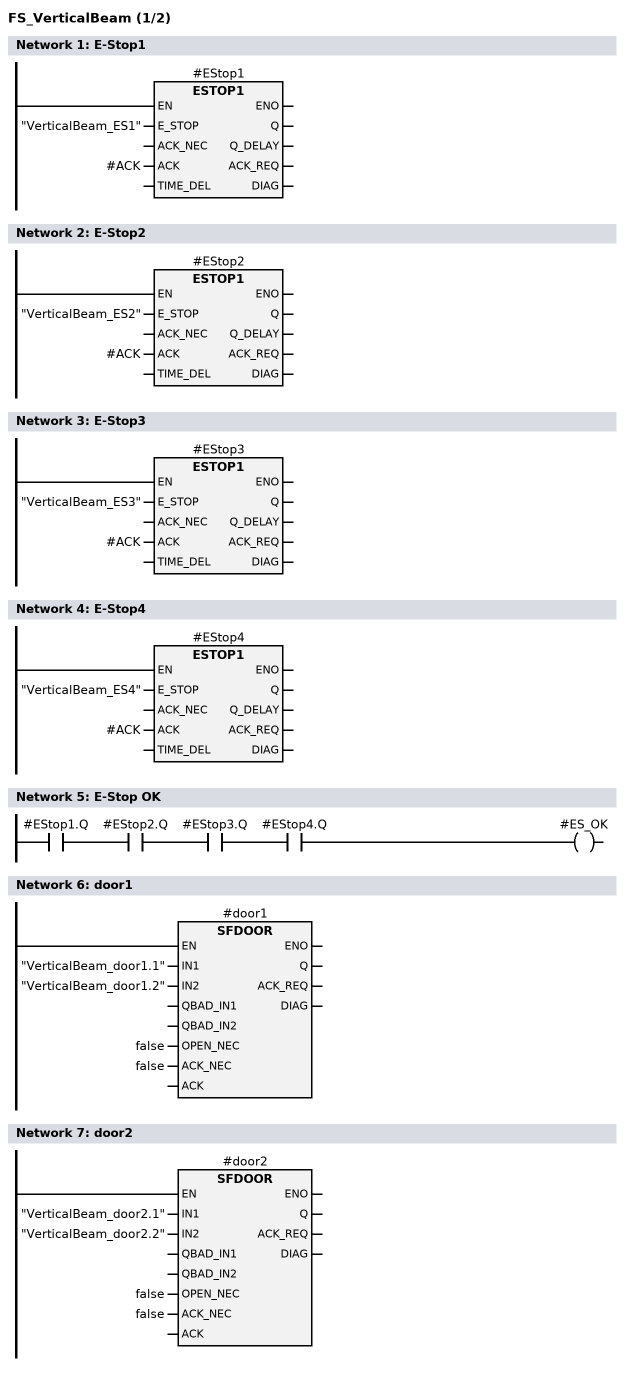
   RUNG wire#powerrail
      #EStop1.ESTOP1(E_STOP := "VerticalBeam_ES1", ACK_NEC :=, ACK := #ACK, TIME_DEL :=, Q =>, Q_DELAY =>, ACK_REQ =>, DIAG =>)
   END_RUNG
   // the same network as SCL:
   #EStop1(E_STOP := "VerticalBeam_ES1", ACK := #ACK);   // ESTOP1
END_REGION

REGION Network 2: E-Stop2
   RUNG wire#powerrail
      #EStop2.ESTOP1(E_STOP := "VerticalBeam_ES2", ACK_NEC :=, ACK := #ACK, TIME_DEL :=, Q =>, Q_DELAY =>, ACK_REQ =>, DIAG =>)
   END_RUNG
   // the same network as SCL:
   #EStop2(E_STOP := "VerticalBeam_ES2", ACK := #ACK);   // ESTOP1
END_REGION

REGION Network 3: E-Stop3
   RUNG wire#powerrail
      #EStop3.ESTOP1(E_STOP := "VerticalBeam_ES3", ACK_NEC :=, ACK := #ACK, TIME_DEL :=, Q =>, Q_DELAY =>, ACK_REQ =>, DIAG =>)
   END_RUNG
   // the same network as SCL:
   #EStop3(E_STOP := "VerticalBeam_ES3", ACK := #ACK);   // ESTOP1
END_REGION

REGION Network 4: E-Stop4
   RUNG wire#powerrail
      #EStop4.ESTOP1(E_STOP := "VerticalBeam_ES4", ACK_NEC :=, ACK := #ACK, TIME_DEL :=, Q =>, Q_DELAY =>, ACK_REQ =>, DIAG =>)
   END_RUNG
   // the same network as SCL:
   #EStop4(E_STOP := "VerticalBeam_ES4", ACK := #ACK);   // ESTOP1
END_REGION

REGION Network 5: E-Stop OK
   RUNG wire#powerrail
      Contact( #EStop1.Q )
      Contact( #EStop2.Q )
      Contact( #EStop3.Q )
      Contact( #EStop4.Q )
      Coil( #ES_OK )
   END_RUNG
   // the same network as SCL:
   #ES_OK := #EStop1.Q AND #EStop2.Q AND #EStop3.Q AND #EStop4.Q;
END_REGION

REGION Network 6: door1
   RUNG wire#powerrail
      #door1.SFDOOR(IN1 := "VerticalBeam_door1.1", IN2 := "VerticalBeam_door1.2", QBAD_IN1 :=, QBAD_IN2 :=, OPEN_NEC := false, ACK_NEC := false, ACK :=, Q =>, ACK_REQ =>, DIAG =>)
   END_RUNG
   // the same network as SCL:
   #door1(IN1 := "VerticalBeam_door1.1", IN2 := "VerticalBeam_door1.2", OPEN_NEC := false, ACK_NEC := false);   // SFDOOR
END_REGION

REGION Network 7: door2
   RUNG wire#powerrail
      #door2.SFDOOR(IN1 := "VerticalBeam_door2.1", IN2 := "VerticalBeam_door2.2", QBAD_IN1 :=, QBAD_IN2 :=, OPEN_NEC := false, ACK_NEC := false, ACK :=, Q =>, ACK_REQ =>, DIAG =>)
   END_RUNG
   // the same network as SCL:
   #door2(IN1 := "VerticalBeam_door2.1", IN2 := "VerticalBeam_door2.2", OPEN_NEC := false, ACK_NEC := false);   // SFDOOR
END_REGION

REGION Network 8: Key
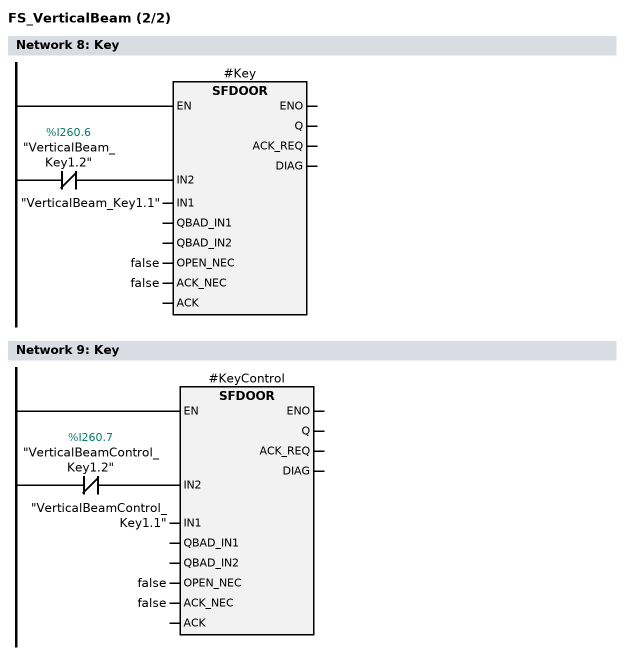
   RUNG wire#powerrail
      #Key.SFDOOR(IN2 := wire#w1, IN1 := "VerticalBeam_Key1.1", QBAD_IN1 :=, QBAD_IN2 :=, OPEN_NEC := false, ACK_NEC := false, ACK :=, Q =>, ACK_REQ =>, DIAG =>)
   END_RUNG
   RUNG wire#powerrail
      I_Contact( "VerticalBeam_Key1.2" )
   END_RUNG wire#w1
   // the same network as SCL:
   #Key(IN2 := NOT "VerticalBeam_Key1.2", IN1 := "VerticalBeam_Key1.1", OPEN_NEC := false, ACK_NEC := false);   // SFDOOR
END_REGION

REGION Network 9: Key
   RUNG wire#powerrail
      #KeyControl.SFDOOR(IN2 := wire#w1, IN1 := "VerticalBeamControl_Key1.1", QBAD_IN1 :=, QBAD_IN2 :=, OPEN_NEC := false, ACK_NEC := false, ACK :=, Q =>, ACK_REQ =>, DIAG =>)
   END_RUNG
   RUNG wire#powerrail
      I_Contact( "VerticalBeamControl_Key1.2" )
   END_RUNG wire#w1
   // the same network as SCL:
   #KeyControl(IN2 := NOT "VerticalBeamControl_Key1.2",   // SFDOOR
               IN1 := "VerticalBeamControl_Key1.1",
               OPEN_NEC := false,
               ACK_NEC := false);
END_REGION
END_FUNCTION_BLOCK

FUNCTION "F_ChannelDia" : Void   // FC2, F_LAD
{ S7_Optimized_Access := 'TRUE' }
VERSION : 0.1
// stored: AutoNumber true, IsIECCheckEnabled false, UDAEnableTagReadback false
   VAR_INPUT
      PASS_OUT : Bool;
      QBAD : Bool;
      ACK_REQ : Bool;
      Channel0_ValueStatus : Bool;
      Channel1_ValueStatus : Bool;
      Channel2_ValueStatus : Bool;
      Channel3_ValueStatus : Bool;
      Channel4_ValueStatus : Bool;
      Channel5_ValueStatus : Bool;
      Channel6_ValueStatus : Bool;
      Channel7_ValueStatus : Bool;
   END_VAR
   VAR_OUTPUT
      FIODia : "FIODia";
   END_VAR
   VAR_TEMP   // added for the SCL form of the ladder/FBD networks
      _w1 : Bool;
   END_VAR
BEGIN

REGION Network 1: 模块钝化
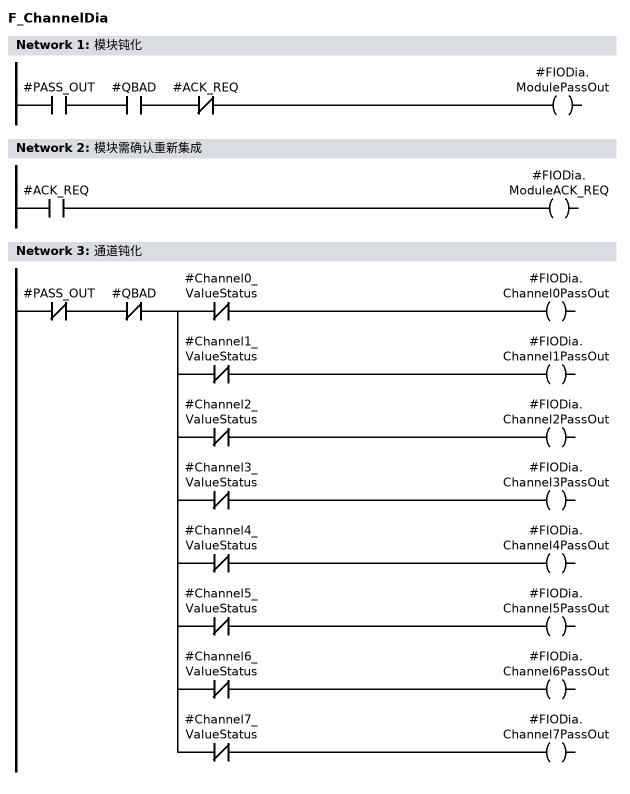
   RUNG wire#powerrail
      Contact( #PASS_OUT )
      Contact( #QBAD )
      I_Contact( #ACK_REQ )
      Coil( #FIODia.ModulePassOut )
   END_RUNG
   // the same network as SCL:
   #FIODia.ModulePassOut := #PASS_OUT AND #QBAD AND NOT #ACK_REQ;
END_REGION

REGION Network 2: 模块需确认重新集成
   RUNG wire#powerrail
      Contact( #ACK_REQ )
      Coil( #FIODia.ModuleACK_REQ )
   END_RUNG
   // the same network as SCL:
   #FIODia.ModuleACK_REQ := #ACK_REQ;
END_REGION

REGION Network 3: 通道钝化
   RUNG wire#powerrail
      I_Contact( #PASS_OUT )
      I_Contact( #QBAD )
      wire#w1
      I_Contact( #Channel0_ValueStatus )
      Coil( #FIODia.Channel0PassOut )
   END_RUNG
   RUNG wire#w1
      I_Contact( #Channel1_ValueStatus )
      Coil( #FIODia.Channel1PassOut )
   END_RUNG
   RUNG wire#w1
      I_Contact( #Channel2_ValueStatus )
      Coil( #FIODia.Channel2PassOut )
   END_RUNG
   RUNG wire#w1
      I_Contact( #Channel3_ValueStatus )
      Coil( #FIODia.Channel3PassOut )
   END_RUNG
   RUNG wire#w1
      I_Contact( #Channel4_ValueStatus )
      Coil( #FIODia.Channel4PassOut )
   END_RUNG
   RUNG wire#w1
      I_Contact( #Channel5_ValueStatus )
      Coil( #FIODia.Channel5PassOut )
   END_RUNG
   RUNG wire#w1
      I_Contact( #Channel6_ValueStatus )
      Coil( #FIODia.Channel6PassOut )
   END_RUNG
   RUNG wire#w1
      I_Contact( #Channel7_ValueStatus )
      Coil( #FIODia.Channel7PassOut )
   END_RUNG
   // the same network as SCL:
   #_w1 := NOT #PASS_OUT AND NOT #QBAD;
   #FIODia.Channel0PassOut := #_w1 AND NOT #Channel0_ValueStatus;
   #FIODia.Channel1PassOut := #_w1 AND NOT #Channel1_ValueStatus;
   #FIODia.Channel2PassOut := #_w1 AND NOT #Channel2_ValueStatus;
   #FIODia.Channel3PassOut := #_w1 AND NOT #Channel3_ValueStatus;
   #FIODia.Channel4PassOut := #_w1 AND NOT #Channel4_ValueStatus;
   #FIODia.Channel5PassOut := #_w1 AND NOT #Channel5_ValueStatus;
   #FIODia.Channel6PassOut := #_w1 AND NOT #Channel6_ValueStatus;
   #FIODia.Channel7PassOut := #_w1 AND NOT #Channel7_ValueStatus;
END_REGION
END_FUNCTION

FUNCTION "Interlock" : Void   // FC1, F_LAD
{ S7_Optimized_Access := 'TRUE' }
VERSION : 0.1
// stored: AutoNumber true, IsIECCheckEnabled false, UDAEnableTagReadback false
   VAR_INPUT
      Room1_Interlock : Bool;
      Room2_Interlock : Bool;
      ACC_Interlock : Bool;
      VerticalBeam_Interlock : Bool;
      "E-stop" : Bool;
   END_VAR
BEGIN

REGION Network 1
   // 暂未考虑模块钝化和通道钝化情况
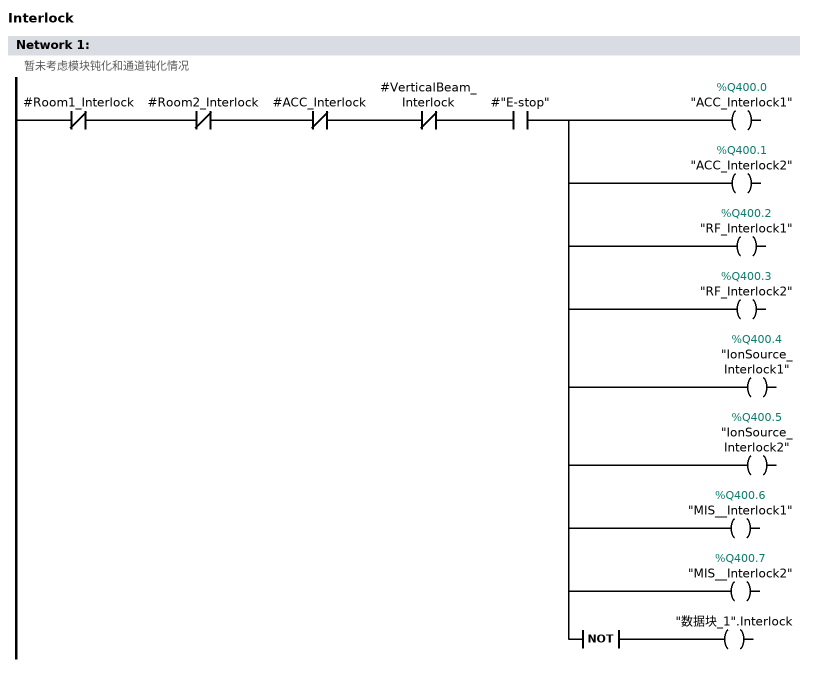
   RUNG wire#powerrail
      I_Contact( #Room1_Interlock )
      I_Contact( #Room2_Interlock )
      I_Contact( #ACC_Interlock )
      I_Contact( #VerticalBeam_Interlock )
      Contact( #"E-stop" )
      wire#w1
      Coil( "ACC_Interlock1" )
   END_RUNG
   RUNG wire#w1
      Coil( "ACC_Interlock2" )
   END_RUNG
   RUNG wire#w1
      Coil( "RF_Interlock1" )
   END_RUNG
   RUNG wire#w1
      Coil( "RF_Interlock2" )
   END_RUNG
   RUNG wire#w1
      Coil( "IonSource_Interlock1" )
   END_RUNG
   RUNG wire#w1
      Coil( "IonSource_Interlock2" )
   END_RUNG
   RUNG wire#w1
      Coil( "MIS__Interlock1" )
   END_RUNG
   RUNG wire#w1
      Coil( "MIS__Interlock2" )
   END_RUNG
   RUNG wire#w1
      Not()
      Coil( "数据块_1".Interlock )
   END_RUNG
   // the same network as SCL:
   "ACC_Interlock1" := NOT #Room1_Interlock AND NOT #Room2_Interlock AND NOT #ACC_Interlock AND NOT #VerticalBeam_Interlock AND #"E-stop";
   "ACC_Interlock2" := "ACC_Interlock1";
   "RF_Interlock1" := "ACC_Interlock1";
   "RF_Interlock2" := "ACC_Interlock1";
   "IonSource_Interlock1" := "ACC_Interlock1";
   "IonSource_Interlock2" := "ACC_Interlock1";
   "MIS__Interlock1" := "ACC_Interlock1";
   "MIS__Interlock2" := "ACC_Interlock1";
   "数据块_1".Interlock := NOT "ACC_Interlock1";
END_REGION
END_FUNCTION

FUNCTION_BLOCK "Main_Safety_RTG1"   // FB1, F_LAD
{ S7_Optimized_Access := 'TRUE' }
VERSION : 0.1
// stored: AutoNumber false, IsIECCheckEnabled false, UDAEnableTagReadback false
   VAR
      ACK_GL_Instance : ACK_GL;
      FS_Room1_Instance : "FS_Room1";
      FS_Room2_Instance : "FS_Room2";
      FS_ACC_Instance : "FS_ACC";
      FS_VerticalBeam_Instance : "FS_VerticalBeam";
   END_VAR
BEGIN

REGION Network 1: 全局确认钝化
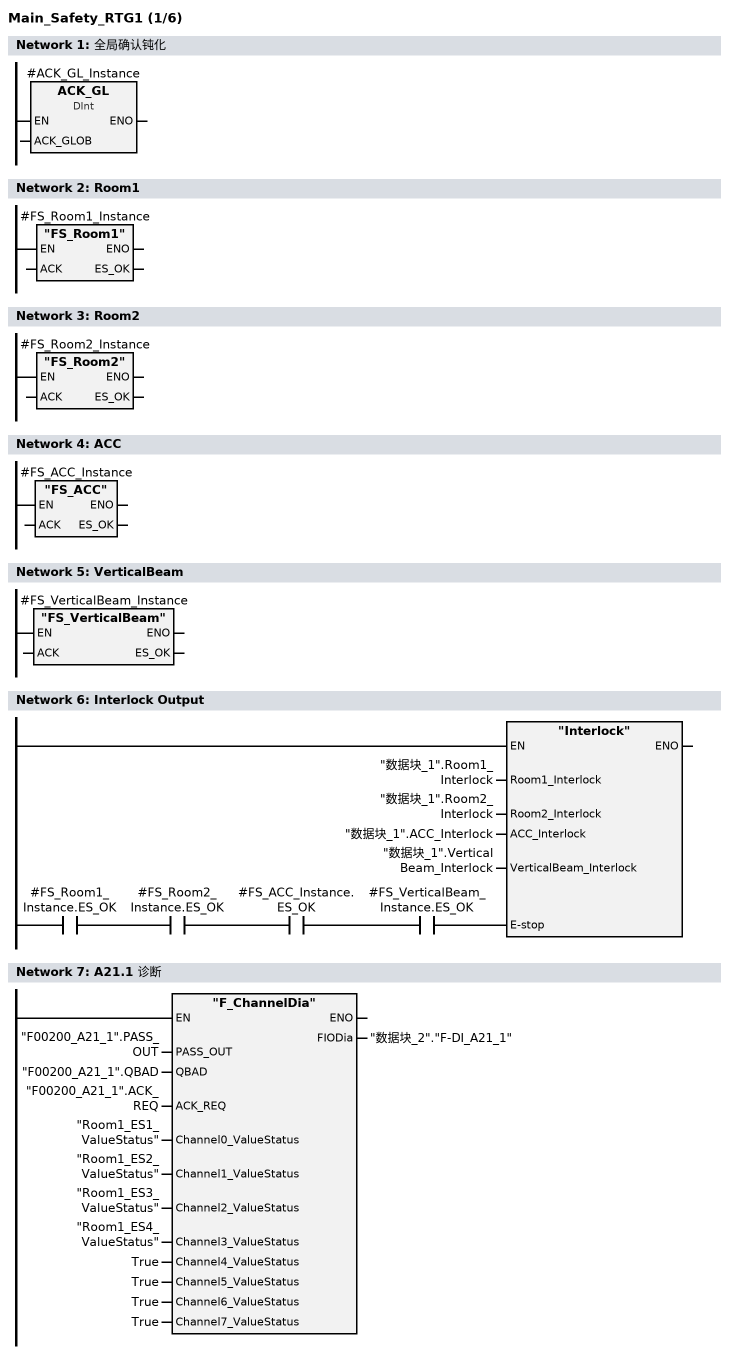
   RUNG wire#powerrail
      { S7_Templates := "codedbool_type := DInt" } #ACK_GL_Instance.ACK_GL(ACK_GLOB :=)
   END_RUNG
   // the same network as SCL:
   #ACK_GL_Instance();   // ACK_GL
END_REGION

REGION Network 2: Room1
   RUNG wire#powerrail
      #FS_Room1_Instance(ACK :=, ES_OK =>)
   END_RUNG
   // the same network as SCL:
   #FS_Room1_Instance();   // "FS_Room1"
END_REGION

REGION Network 3: Room2
   RUNG wire#powerrail
      #FS_Room2_Instance(ACK :=, ES_OK =>)
   END_RUNG
   // the same network as SCL:
   #FS_Room2_Instance();   // "FS_Room2"
END_REGION

REGION Network 4: ACC
   RUNG wire#powerrail
      #FS_ACC_Instance(ACK :=, ES_OK =>)
   END_RUNG
   // the same network as SCL:
   #FS_ACC_Instance();   // "FS_ACC"
END_REGION

REGION Network 5: VerticalBeam
   RUNG wire#powerrail
      #FS_VerticalBeam_Instance(ACK :=, ES_OK =>)
   END_RUNG
   // the same network as SCL:
   #FS_VerticalBeam_Instance();   // "FS_VerticalBeam"
END_REGION

REGION Network 6: Interlock Output
   RUNG wire#powerrail
      "Interlock"(Room1_Interlock := "数据块_1".Room1_Interlock, Room2_Interlock := "数据块_1".Room2_Interlock, ACC_Interlock := "数据块_1".ACC_Interlock, VerticalBeam_Interlock := "数据块_1".VerticalBeam_Interlock, "E-stop" := wire#w1)
   END_RUNG
   RUNG wire#powerrail
      Contact( #FS_Room1_Instance.ES_OK )
      Contact( #FS_Room2_Instance.ES_OK )
      Contact( #FS_ACC_Instance.ES_OK )
      Contact( #FS_VerticalBeam_Instance.ES_OK )
   END_RUNG wire#w1
   // the same network as SCL:
   "Interlock"(Room1_Interlock := "数据块_1".Room1_Interlock,
               Room2_Interlock := "数据块_1".Room2_Interlock,
               ACC_Interlock := "数据块_1".ACC_Interlock,
               VerticalBeam_Interlock := "数据块_1".VerticalBeam_Interlock,
               "E-stop" := #FS_Room1_Instance.ES_OK AND #FS_Room2_Instance.ES_OK AND #FS_ACC_Instance.ES_OK AND #FS_VerticalBeam_Instance.ES_OK);
END_REGION

REGION Network 7: A21.1 诊断
   RUNG wire#powerrail
      "F_ChannelDia"(PASS_OUT := "F00200_A21_1".PASS_OUT, QBAD := "F00200_A21_1".QBAD, ACK_REQ := "F00200_A21_1".ACK_REQ, Channel0_ValueStatus := "Room1_ES1_ValueStatus", Channel1_ValueStatus := "Room1_ES2_ValueStatus", Channel2_ValueStatus := "Room1_ES3_ValueStatus", Channel3_ValueStatus := "Room1_ES4_ValueStatus", Channel4_ValueStatus := True, Channel5_ValueStatus := True, Channel6_ValueStatus := True, Channel7_ValueStatus := True, FIODia => "数据块_2"."F-DI_A21_1")
   END_RUNG
   // the same network as SCL:
   "F_ChannelDia"(PASS_OUT := "F00200_A21_1".PASS_OUT,
                  QBAD := "F00200_A21_1".QBAD,
                  ACK_REQ := "F00200_A21_1".ACK_REQ,
                  Channel0_ValueStatus := "Room1_ES1_ValueStatus",
                  Channel1_ValueStatus := "Room1_ES2_ValueStatus",
                  Channel2_ValueStatus := "Room1_ES3_ValueStatus",
                  Channel3_ValueStatus := "Room1_ES4_ValueStatus",
                  Channel4_ValueStatus := True,
                  Channel5_ValueStatus := True,
                  Channel6_ValueStatus := True,
                  Channel7_ValueStatus := True,
                  FIODia => "数据块_2"."F-DI_A21_1");
END_REGION

REGION Network 8: A21.2 诊断
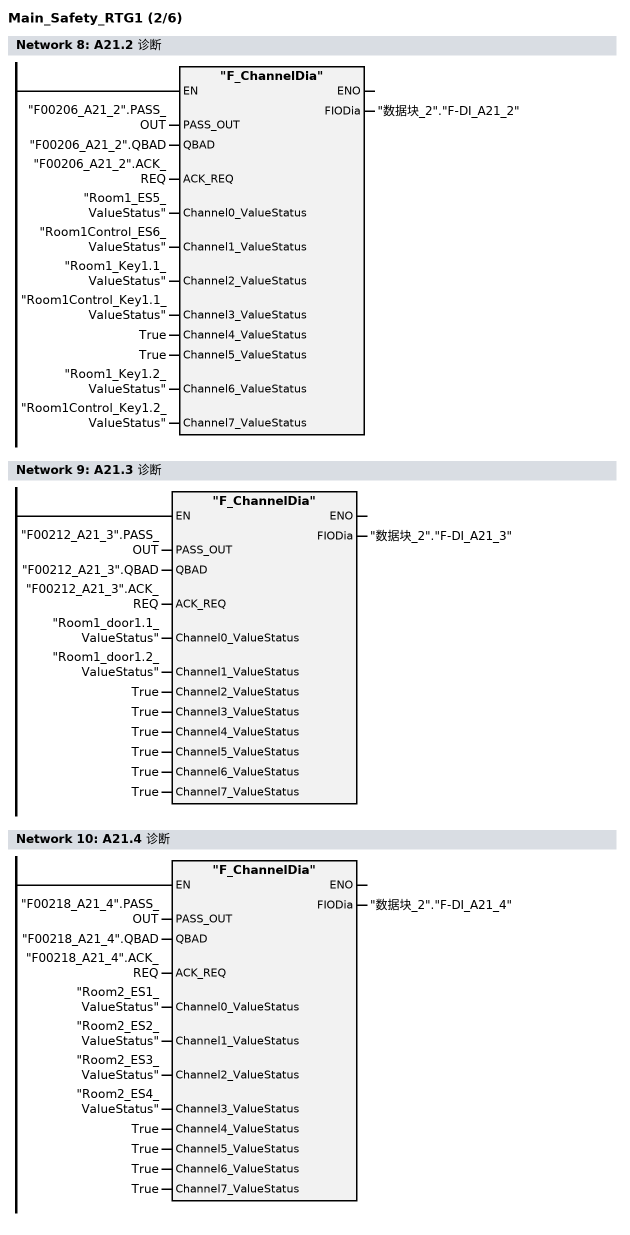
   RUNG wire#powerrail
      "F_ChannelDia"(PASS_OUT := "F00206_A21_2".PASS_OUT, QBAD := "F00206_A21_2".QBAD, ACK_REQ := "F00206_A21_2".ACK_REQ, Channel0_ValueStatus := "Room1_ES5_ValueStatus", Channel1_ValueStatus := "Room1Control_ES6_ValueStatus", Channel2_ValueStatus := "Room1_Key1.1_ValueStatus", Channel3_ValueStatus := "Room1Control_Key1.1_ValueStatus", Channel4_ValueStatus := True, Channel5_ValueStatus := True, Channel6_ValueStatus := "Room1_Key1.2_ValueStatus", Channel7_ValueStatus := "Room1Control_Key1.2_ValueStatus", FIODia => "数据块_2"."F-DI_A21_2")
   END_RUNG
   // the same network as SCL:
   "F_ChannelDia"(PASS_OUT := "F00206_A21_2".PASS_OUT,
                  QBAD := "F00206_A21_2".QBAD,
                  ACK_REQ := "F00206_A21_2".ACK_REQ,
                  Channel0_ValueStatus := "Room1_ES5_ValueStatus",
                  Channel1_ValueStatus := "Room1Control_ES6_ValueStatus",
                  Channel2_ValueStatus := "Room1_Key1.1_ValueStatus",
                  Channel3_ValueStatus := "Room1Control_Key1.1_ValueStatus",
                  Channel4_ValueStatus := True,
                  Channel5_ValueStatus := True,
                  Channel6_ValueStatus := "Room1_Key1.2_ValueStatus",
                  Channel7_ValueStatus := "Room1Control_Key1.2_ValueStatus",
                  FIODia => "数据块_2"."F-DI_A21_2");
END_REGION

REGION Network 9: A21.3 诊断
   RUNG wire#powerrail
      "F_ChannelDia"(PASS_OUT := "F00212_A21_3".PASS_OUT, QBAD := "F00212_A21_3".QBAD, ACK_REQ := "F00212_A21_3".ACK_REQ, Channel0_ValueStatus := "Room1_door1.1_ValueStatus", Channel1_ValueStatus := "Room1_door1.2_ValueStatus", Channel2_ValueStatus := True, Channel3_ValueStatus := True, Channel4_ValueStatus := True, Channel5_ValueStatus := True, Channel6_ValueStatus := True, Channel7_ValueStatus := True, FIODia => "数据块_2"."F-DI_A21_3")
   END_RUNG
   // the same network as SCL:
   "F_ChannelDia"(PASS_OUT := "F00212_A21_3".PASS_OUT,
                  QBAD := "F00212_A21_3".QBAD,
                  ACK_REQ := "F00212_A21_3".ACK_REQ,
                  Channel0_ValueStatus := "Room1_door1.1_ValueStatus",
                  Channel1_ValueStatus := "Room1_door1.2_ValueStatus",
                  Channel2_ValueStatus := True,
                  Channel3_ValueStatus := True,
                  Channel4_ValueStatus := True,
                  Channel5_ValueStatus := True,
                  Channel6_ValueStatus := True,
                  Channel7_ValueStatus := True,
                  FIODia => "数据块_2"."F-DI_A21_3");
END_REGION

REGION Network 10: A21.4 诊断
   RUNG wire#powerrail
      "F_ChannelDia"(PASS_OUT := "F00218_A21_4".PASS_OUT, QBAD := "F00218_A21_4".QBAD, ACK_REQ := "F00218_A21_4".ACK_REQ, Channel0_ValueStatus := "Room2_ES1_ValueStatus", Channel1_ValueStatus := "Room2_ES2_ValueStatus", Channel2_ValueStatus := "Room2_ES3_ValueStatus", Channel3_ValueStatus := "Room2_ES4_ValueStatus", Channel4_ValueStatus := True, Channel5_ValueStatus := True, Channel6_ValueStatus := True, Channel7_ValueStatus := True, FIODia => "数据块_2"."F-DI_A21_4")
   END_RUNG
   // the same network as SCL:
   "F_ChannelDia"(PASS_OUT := "F00218_A21_4".PASS_OUT,
                  QBAD := "F00218_A21_4".QBAD,
                  ACK_REQ := "F00218_A21_4".ACK_REQ,
                  Channel0_ValueStatus := "Room2_ES1_ValueStatus",
                  Channel1_ValueStatus := "Room2_ES2_ValueStatus",
                  Channel2_ValueStatus := "Room2_ES3_ValueStatus",
                  Channel3_ValueStatus := "Room2_ES4_ValueStatus",
                  Channel4_ValueStatus := True,
                  Channel5_ValueStatus := True,
                  Channel6_ValueStatus := True,
                  Channel7_ValueStatus := True,
                  FIODia => "数据块_2"."F-DI_A21_4");
END_REGION

REGION Network 11: A21.5 诊断
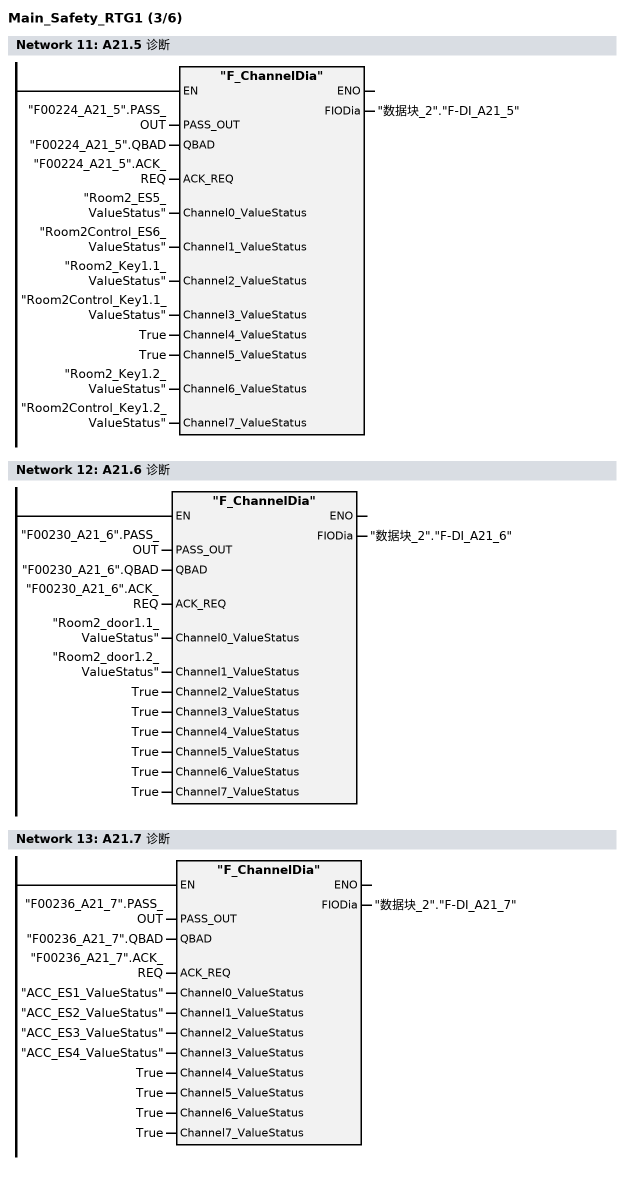
   RUNG wire#powerrail
      "F_ChannelDia"(PASS_OUT := "F00224_A21_5".PASS_OUT, QBAD := "F00224_A21_5".QBAD, ACK_REQ := "F00224_A21_5".ACK_REQ, Channel0_ValueStatus := "Room2_ES5_ValueStatus", Channel1_ValueStatus := "Room2Control_ES6_ValueStatus", Channel2_ValueStatus := "Room2_Key1.1_ValueStatus", Channel3_ValueStatus := "Room2Control_Key1.1_ValueStatus", Channel4_ValueStatus := True, Channel5_ValueStatus := True, Channel6_ValueStatus := "Room2_Key1.2_ValueStatus", Channel7_ValueStatus := "Room2Control_Key1.2_ValueStatus", FIODia => "数据块_2"."F-DI_A21_5")
   END_RUNG
   // the same network as SCL:
   "F_ChannelDia"(PASS_OUT := "F00224_A21_5".PASS_OUT,
                  QBAD := "F00224_A21_5".QBAD,
                  ACK_REQ := "F00224_A21_5".ACK_REQ,
                  Channel0_ValueStatus := "Room2_ES5_ValueStatus",
                  Channel1_ValueStatus := "Room2Control_ES6_ValueStatus",
                  Channel2_ValueStatus := "Room2_Key1.1_ValueStatus",
                  Channel3_ValueStatus := "Room2Control_Key1.1_ValueStatus",
                  Channel4_ValueStatus := True,
                  Channel5_ValueStatus := True,
                  Channel6_ValueStatus := "Room2_Key1.2_ValueStatus",
                  Channel7_ValueStatus := "Room2Control_Key1.2_ValueStatus",
                  FIODia => "数据块_2"."F-DI_A21_5");
END_REGION

REGION Network 12: A21.6 诊断
   RUNG wire#powerrail
      "F_ChannelDia"(PASS_OUT := "F00230_A21_6".PASS_OUT, QBAD := "F00230_A21_6".QBAD, ACK_REQ := "F00230_A21_6".ACK_REQ, Channel0_ValueStatus := "Room2_door1.1_ValueStatus", Channel1_ValueStatus := "Room2_door1.2_ValueStatus", Channel2_ValueStatus := True, Channel3_ValueStatus := True, Channel4_ValueStatus := True, Channel5_ValueStatus := True, Channel6_ValueStatus := True, Channel7_ValueStatus := True, FIODia => "数据块_2"."F-DI_A21_6")
   END_RUNG
   // the same network as SCL:
   "F_ChannelDia"(PASS_OUT := "F00230_A21_6".PASS_OUT,
                  QBAD := "F00230_A21_6".QBAD,
                  ACK_REQ := "F00230_A21_6".ACK_REQ,
                  Channel0_ValueStatus := "Room2_door1.1_ValueStatus",
                  Channel1_ValueStatus := "Room2_door1.2_ValueStatus",
                  Channel2_ValueStatus := True,
                  Channel3_ValueStatus := True,
                  Channel4_ValueStatus := True,
                  Channel5_ValueStatus := True,
                  Channel6_ValueStatus := True,
                  Channel7_ValueStatus := True,
                  FIODia => "数据块_2"."F-DI_A21_6");
END_REGION

REGION Network 13: A21.7 诊断
   RUNG wire#powerrail
      "F_ChannelDia"(PASS_OUT := "F00236_A21_7".PASS_OUT, QBAD := "F00236_A21_7".QBAD, ACK_REQ := "F00236_A21_7".ACK_REQ, Channel0_ValueStatus := "ACC_ES1_ValueStatus", Channel1_ValueStatus := "ACC_ES2_ValueStatus", Channel2_ValueStatus := "ACC_ES3_ValueStatus", Channel3_ValueStatus := "ACC_ES4_ValueStatus", Channel4_ValueStatus := True, Channel5_ValueStatus := True, Channel6_ValueStatus := True, Channel7_ValueStatus := True, FIODia => "数据块_2"."F-DI_A21_7")
   END_RUNG
   // the same network as SCL:
   "F_ChannelDia"(PASS_OUT := "F00236_A21_7".PASS_OUT,
                  QBAD := "F00236_A21_7".QBAD,
                  ACK_REQ := "F00236_A21_7".ACK_REQ,
                  Channel0_ValueStatus := "ACC_ES1_ValueStatus",
                  Channel1_ValueStatus := "ACC_ES2_ValueStatus",
                  Channel2_ValueStatus := "ACC_ES3_ValueStatus",
                  Channel3_ValueStatus := "ACC_ES4_ValueStatus",
                  Channel4_ValueStatus := True,
                  Channel5_ValueStatus := True,
                  Channel6_ValueStatus := True,
                  Channel7_ValueStatus := True,
                  FIODia => "数据块_2"."F-DI_A21_7");
END_REGION

REGION Network 14: A21.8 诊断
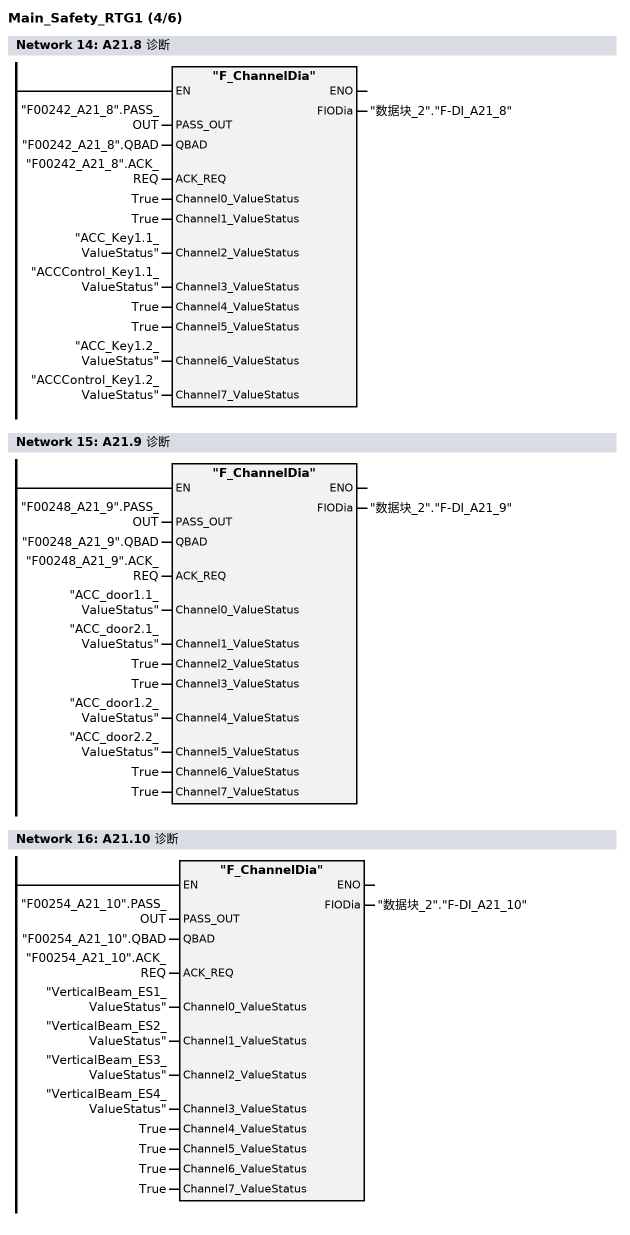
   RUNG wire#powerrail
      "F_ChannelDia"(PASS_OUT := "F00242_A21_8".PASS_OUT, QBAD := "F00242_A21_8".QBAD, ACK_REQ := "F00242_A21_8".ACK_REQ, Channel0_ValueStatus := True, Channel1_ValueStatus := True, Channel2_ValueStatus := "ACC_Key1.1_ValueStatus", Channel3_ValueStatus := "ACCControl_Key1.1_ValueStatus", Channel4_ValueStatus := True, Channel5_ValueStatus := True, Channel6_ValueStatus := "ACC_Key1.2_ValueStatus", Channel7_ValueStatus := "ACCControl_Key1.2_ValueStatus", FIODia => "数据块_2"."F-DI_A21_8")
   END_RUNG
   // the same network as SCL:
   "F_ChannelDia"(PASS_OUT := "F00242_A21_8".PASS_OUT,
                  QBAD := "F00242_A21_8".QBAD,
                  ACK_REQ := "F00242_A21_8".ACK_REQ,
                  Channel0_ValueStatus := True,
                  Channel1_ValueStatus := True,
                  Channel2_ValueStatus := "ACC_Key1.1_ValueStatus",
                  Channel3_ValueStatus := "ACCControl_Key1.1_ValueStatus",
                  Channel4_ValueStatus := True,
                  Channel5_ValueStatus := True,
                  Channel6_ValueStatus := "ACC_Key1.2_ValueStatus",
                  Channel7_ValueStatus := "ACCControl_Key1.2_ValueStatus",
                  FIODia => "数据块_2"."F-DI_A21_8");
END_REGION

REGION Network 15: A21.9 诊断
   RUNG wire#powerrail
      "F_ChannelDia"(PASS_OUT := "F00248_A21_9".PASS_OUT, QBAD := "F00248_A21_9".QBAD, ACK_REQ := "F00248_A21_9".ACK_REQ, Channel0_ValueStatus := "ACC_door1.1_ValueStatus", Channel1_ValueStatus := "ACC_door2.1_ValueStatus", Channel2_ValueStatus := True, Channel3_ValueStatus := True, Channel4_ValueStatus := "ACC_door1.2_ValueStatus", Channel5_ValueStatus := "ACC_door2.2_ValueStatus", Channel6_ValueStatus := True, Channel7_ValueStatus := True, FIODia => "数据块_2"."F-DI_A21_9")
   END_RUNG
   // the same network as SCL:
   "F_ChannelDia"(PASS_OUT := "F00248_A21_9".PASS_OUT,
                  QBAD := "F00248_A21_9".QBAD,
                  ACK_REQ := "F00248_A21_9".ACK_REQ,
                  Channel0_ValueStatus := "ACC_door1.1_ValueStatus",
                  Channel1_ValueStatus := "ACC_door2.1_ValueStatus",
                  Channel2_ValueStatus := True,
                  Channel3_ValueStatus := True,
                  Channel4_ValueStatus := "ACC_door1.2_ValueStatus",
                  Channel5_ValueStatus := "ACC_door2.2_ValueStatus",
                  Channel6_ValueStatus := True,
                  Channel7_ValueStatus := True,
                  FIODia => "数据块_2"."F-DI_A21_9");
END_REGION

REGION Network 16: A21.10 诊断
   RUNG wire#powerrail
      "F_ChannelDia"(PASS_OUT := "F00254_A21_10".PASS_OUT, QBAD := "F00254_A21_10".QBAD, ACK_REQ := "F00254_A21_10".ACK_REQ, Channel0_ValueStatus := "VerticalBeam_ES1_ValueStatus", Channel1_ValueStatus := "VerticalBeam_ES2_ValueStatus", Channel2_ValueStatus := "VerticalBeam_ES3_ValueStatus", Channel3_ValueStatus := "VerticalBeam_ES4_ValueStatus", Channel4_ValueStatus := True, Channel5_ValueStatus := True, Channel6_ValueStatus := True, Channel7_ValueStatus := True, FIODia => "数据块_2"."F-DI_A21_10")
   END_RUNG
   // the same network as SCL:
   "F_ChannelDia"(PASS_OUT := "F00254_A21_10".PASS_OUT,
                  QBAD := "F00254_A21_10".QBAD,
                  ACK_REQ := "F00254_A21_10".ACK_REQ,
                  Channel0_ValueStatus := "VerticalBeam_ES1_ValueStatus",
                  Channel1_ValueStatus := "VerticalBeam_ES2_ValueStatus",
                  Channel2_ValueStatus := "VerticalBeam_ES3_ValueStatus",
                  Channel3_ValueStatus := "VerticalBeam_ES4_ValueStatus",
                  Channel4_ValueStatus := True,
                  Channel5_ValueStatus := True,
                  Channel6_ValueStatus := True,
                  Channel7_ValueStatus := True,
                  FIODia => "数据块_2"."F-DI_A21_10");
END_REGION

REGION Network 17: A21.11 诊断
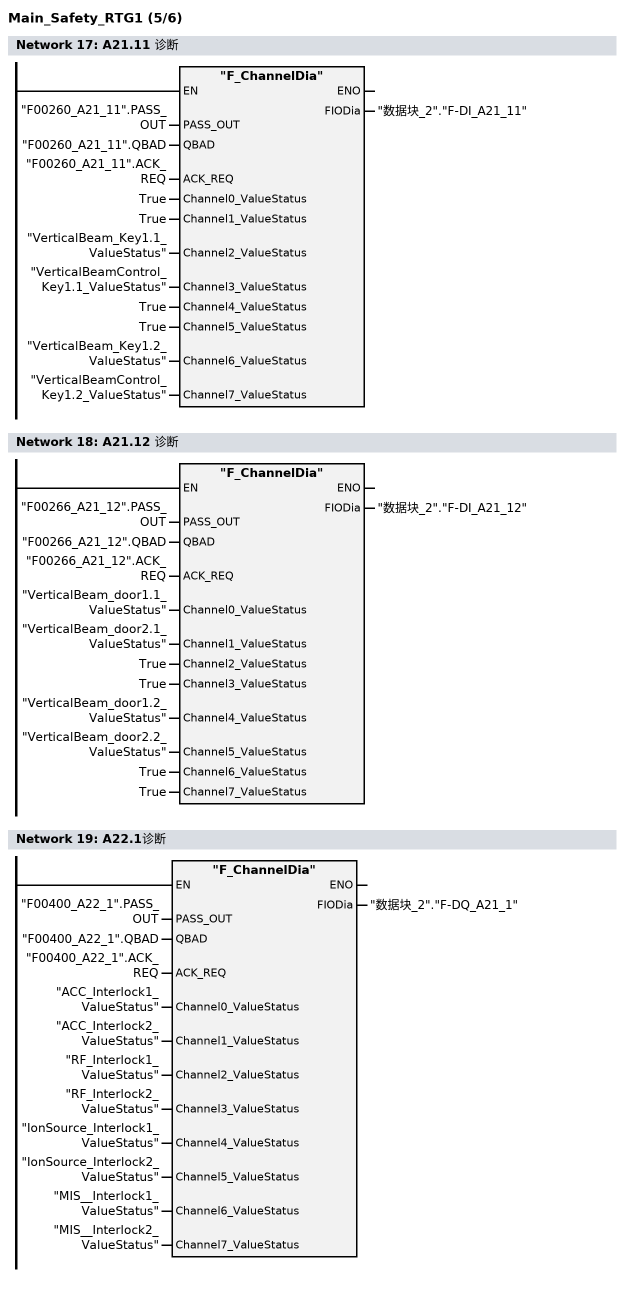
   RUNG wire#powerrail
      "F_ChannelDia"(PASS_OUT := "F00260_A21_11".PASS_OUT, QBAD := "F00260_A21_11".QBAD, ACK_REQ := "F00260_A21_11".ACK_REQ, Channel0_ValueStatus := True, Channel1_ValueStatus := True, Channel2_ValueStatus := "VerticalBeam_Key1.1_ValueStatus", Channel3_ValueStatus := "VerticalBeamControl_Key1.1_ValueStatus", Channel4_ValueStatus := True, Channel5_ValueStatus := True, Channel6_ValueStatus := "VerticalBeam_Key1.2_ValueStatus", Channel7_ValueStatus := "VerticalBeamControl_Key1.2_ValueStatus", FIODia => "数据块_2"."F-DI_A21_11")
   END_RUNG
   // the same network as SCL:
   "F_ChannelDia"(PASS_OUT := "F00260_A21_11".PASS_OUT,
                  QBAD := "F00260_A21_11".QBAD,
                  ACK_REQ := "F00260_A21_11".ACK_REQ,
                  Channel0_ValueStatus := True,
                  Channel1_ValueStatus := True,
                  Channel2_ValueStatus := "VerticalBeam_Key1.1_ValueStatus",
                  Channel3_ValueStatus := "VerticalBeamControl_Key1.1_ValueStatus",
                  Channel4_ValueStatus := True,
                  Channel5_ValueStatus := True,
                  Channel6_ValueStatus := "VerticalBeam_Key1.2_ValueStatus",
                  Channel7_ValueStatus := "VerticalBeamControl_Key1.2_ValueStatus",
                  FIODia => "数据块_2"."F-DI_A21_11");
END_REGION

REGION Network 18: A21.12 诊断
   RUNG wire#powerrail
      "F_ChannelDia"(PASS_OUT := "F00266_A21_12".PASS_OUT, QBAD := "F00266_A21_12".QBAD, ACK_REQ := "F00266_A21_12".ACK_REQ, Channel0_ValueStatus := "VerticalBeam_door1.1_ValueStatus", Channel1_ValueStatus := "VerticalBeam_door2.1_ValueStatus", Channel2_ValueStatus := True, Channel3_ValueStatus := True, Channel4_ValueStatus := "VerticalBeam_door1.2_ValueStatus", Channel5_ValueStatus := "VerticalBeam_door2.2_ValueStatus", Channel6_ValueStatus := True, Channel7_ValueStatus := True, FIODia => "数据块_2"."F-DI_A21_12")
   END_RUNG
   // the same network as SCL:
   "F_ChannelDia"(PASS_OUT := "F00266_A21_12".PASS_OUT,
                  QBAD := "F00266_A21_12".QBAD,
                  ACK_REQ := "F00266_A21_12".ACK_REQ,
                  Channel0_ValueStatus := "VerticalBeam_door1.1_ValueStatus",
                  Channel1_ValueStatus := "VerticalBeam_door2.1_ValueStatus",
                  Channel2_ValueStatus := True,
                  Channel3_ValueStatus := True,
                  Channel4_ValueStatus := "VerticalBeam_door1.2_ValueStatus",
                  Channel5_ValueStatus := "VerticalBeam_door2.2_ValueStatus",
                  Channel6_ValueStatus := True,
                  Channel7_ValueStatus := True,
                  FIODia => "数据块_2"."F-DI_A21_12");
END_REGION

REGION Network 19: A22.1诊断
   RUNG wire#powerrail
      "F_ChannelDia"(PASS_OUT := "F00400_A22_1".PASS_OUT, QBAD := "F00400_A22_1".QBAD, ACK_REQ := "F00400_A22_1".ACK_REQ, Channel0_ValueStatus := "ACC_Interlock1_ValueStatus", Channel1_ValueStatus := "ACC_Interlock2_ValueStatus", Channel2_ValueStatus := "RF_Interlock1_ValueStatus", Channel3_ValueStatus := "RF_Interlock2_ValueStatus", Channel4_ValueStatus := "IonSource_Interlock1_ValueStatus", Channel5_ValueStatus := "IonSource_Interlock2_ValueStatus", Channel6_ValueStatus := "MIS__Interlock1_ValueStatus", Channel7_ValueStatus := "MIS__Interlock2_ValueStatus", FIODia => "数据块_2"."F-DQ_A21_1")
   END_RUNG
   // the same network as SCL:
   "F_ChannelDia"(PASS_OUT := "F00400_A22_1".PASS_OUT,
                  QBAD := "F00400_A22_1".QBAD,
                  ACK_REQ := "F00400_A22_1".ACK_REQ,
                  Channel0_ValueStatus := "ACC_Interlock1_ValueStatus",
                  Channel1_ValueStatus := "ACC_Interlock2_ValueStatus",
                  Channel2_ValueStatus := "RF_Interlock1_ValueStatus",
                  Channel3_ValueStatus := "RF_Interlock2_ValueStatus",
                  Channel4_ValueStatus := "IonSource_Interlock1_ValueStatus",
                  Channel5_ValueStatus := "IonSource_Interlock2_ValueStatus",
                  Channel6_ValueStatus := "MIS__Interlock1_ValueStatus",
                  Channel7_ValueStatus := "MIS__Interlock2_ValueStatus",
                  FIODia => "数据块_2"."F-DQ_A21_1");
END_REGION

REGION Network 20: A22.2诊断
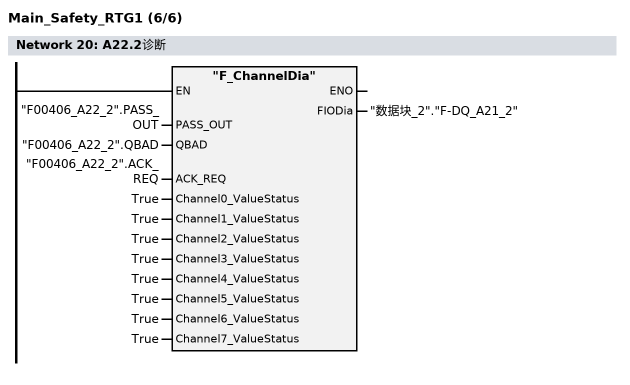
   RUNG wire#powerrail
      "F_ChannelDia"(PASS_OUT := "F00406_A22_2".PASS_OUT, QBAD := "F00406_A22_2".QBAD, ACK_REQ := "F00406_A22_2".ACK_REQ, Channel0_ValueStatus := True, Channel1_ValueStatus := True, Channel2_ValueStatus := True, Channel3_ValueStatus := True, Channel4_ValueStatus := True, Channel5_ValueStatus := True, Channel6_ValueStatus := True, Channel7_ValueStatus := True, FIODia => "数据块_2"."F-DQ_A21_2")
   END_RUNG
   // the same network as SCL:
   "F_ChannelDia"(PASS_OUT := "F00406_A22_2".PASS_OUT,
                  QBAD := "F00406_A22_2".QBAD,
                  ACK_REQ := "F00406_A22_2".ACK_REQ,
                  Channel0_ValueStatus := True,
                  Channel1_ValueStatus := True,
                  Channel2_ValueStatus := True,
                  Channel3_ValueStatus := True,
                  Channel4_ValueStatus := True,
                  Channel5_ValueStatus := True,
                  Channel6_ValueStatus := True,
                  Channel7_ValueStatus := True,
                  FIODia => "数据块_2"."F-DQ_A21_2");
END_REGION
END_FUNCTION_BLOCK

FUNCTION "TCS" : Void   // FC3, LAD
{ S7_Optimized_Access := 'TRUE' }
VERSION : 0.1
// stored: AutoNumber true, IsIECCheckEnabled false, SetENOAutomatically false, UDAEnableTagReadback false
BEGIN

REGION Network 1
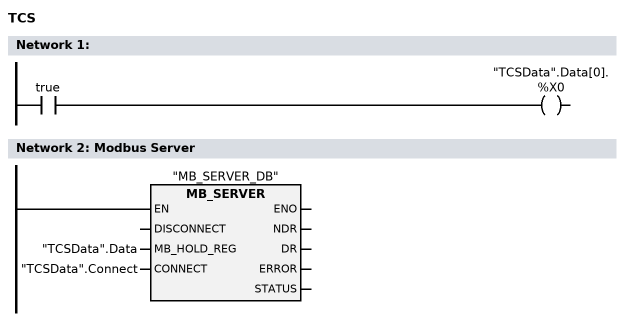
   RUNG wire#powerrail
      Contact( true )
      Coil( "TCSData".Data[0].%X0 )
   END_RUNG
   // the same network as SCL:
   "TCSData".Data[0].%X0 := true;
END_REGION

REGION Network 2: Modbus Server
   RUNG wire#powerrail
      "MB_SERVER_DB".MB_SERVER(DISCONNECT :=, MB_HOLD_REG := "TCSData".Data, CONNECT := "TCSData".Connect, NDR =>, DR =>, ERROR =>, STATUS =>)
   END_RUNG
   // the same network as SCL:
   "MB_SERVER_DB"(MB_HOLD_REG := "TCSData".Data, CONNECT := "TCSData".Connect);   // MB_SERVER
END_REGION
END_FUNCTION

DATA_BLOCK "Main_Safety_RTG1_DB"   // DB1, F_DB
NAME : FUSI
VERSION : 0.1
// stored: AutoNumber true, DBAccessibleFromOPCUA true, InstanceOfName Main_Safety_RTG1, InstanceOfType FB
"Main_Safety_RTG1"
BEGIN
END_DATA_BLOCK

DATA_BLOCK "Room1_AccessControl_idb"   // DB9
VERSION : 0.1
// stored: AutoNumber true, DBAccessibleFromOPCUA true, InstanceOfName AccessControl, InstanceOfType FB
"AccessControl"
BEGIN
END_DATA_BLOCK

DATA_BLOCK "Room1_SearchArea_idb"   // DB6
VERSION : 0.1
// stored: AutoNumber true, DBAccessibleFromOPCUA true, InstanceOfName SearchArea, InstanceOfType FB
"SearchArea"
BEGIN
END_DATA_BLOCK

DATA_BLOCK "Room2_AccessControl_idb"   // DB10
VERSION : 0.1
// stored: AutoNumber true, DBAccessibleFromOPCUA true, InstanceOfName AccessControl, InstanceOfType FB
"AccessControl"
BEGIN
END_DATA_BLOCK

DATA_BLOCK "Room2_SearchArea_idb"   // DB7
VERSION : 0.1
// stored: AutoNumber true, DBAccessibleFromOPCUA true, InstanceOfName SearchArea, InstanceOfType FB
"SearchArea"
BEGIN
END_DATA_BLOCK

DATA_BLOCK "ACC_AccessControl_idb"   // DB12
VERSION : 0.1
// stored: AutoNumber true, DBAccessibleFromOPCUA true, InstanceOfName AccessControl, InstanceOfType FB
"AccessControl"
BEGIN
END_DATA_BLOCK

DATA_BLOCK "ACC_SearchArea_idb"   // DB11
VERSION : 0.1
// stored: AutoNumber true, DBAccessibleFromOPCUA true, InstanceOfName SearchArea_2doors, InstanceOfType FB
"SearchArea_2doors"
BEGIN
END_DATA_BLOCK

DATA_BLOCK "VerticalBeam_AccessControl_idb"   // DB14
VERSION : 0.1
// stored: AutoNumber true, DBAccessibleFromOPCUA true, InstanceOfName AccessControl, InstanceOfType FB
"AccessControl"
BEGIN
END_DATA_BLOCK

DATA_BLOCK "VerticalBeam_SearchArea_idb"   // DB13
VERSION : 0.1
// stored: AutoNumber true, DBAccessibleFromOPCUA true, InstanceOfName SearchArea_2doors, InstanceOfType FB
"SearchArea_2doors"
BEGIN
END_DATA_BLOCK

DATA_BLOCK "MB_SERVER_DB"   // DB5
// stored: AutoNumber true, DBAccessibleFromOPCUA true, InstanceOfName MB_SERVER, OfSystemLibElement MB_SERVER, OfSystemLibVersion 5.3
"MB_SERVER"
   // VAR_INPUT
   //    DISCONNECT { ExternalVisible := 'False'} : Bool;
   // END_VAR
   // VAR_OUTPUT
   //    NDR { ExternalVisible := 'False'} : Bool;
   //    DR { ExternalVisible := 'False'} : Bool;
   //    ERROR { ExternalVisible := 'False'} : Bool;
   //    STATUS { ExternalVisible := 'False'} : Word;
   // END_VAR
   // VAR_IN_OUT
   //    MB_HOLD_REG : Variant;
   //    CONNECT : Variant;
   // END_VAR
   // VAR
   //    TCON { S7_SetPoint := 'True'} : TCON;
   //    TSEND { S7_SetPoint := 'True'} : TSEND;
   //    TRCV { S7_SetPoint := 'True'} : TRCV;
   //    TDIAG { S7_SetPoint := 'True'} : T_DIAG;
   //    TRESET { S7_SetPoint := 'True'} : T_RESET;
   //    TDISCON { S7_SetPoint := 'True'} : TDISCON;
   //    TDIAG_Status { S7_SetPoint := 'True'} : TDiag_Status;
   //    HR_Start_Offset : Word;
   //    QB_Start : UInt;
   //    QB_Count : UInt;
   //    QB_Read_Start : UInt;
   //    QB_Read_Count : UInt;
   //    IB_Read_Start : UInt;
   //    IB_Read_Count : UInt;
   //    Success_Count : Word;
   //    Request_Count : Word;
   //    Xmt_Rcv_Count : Word;
   //    Server_Message_Count : Word;
   //    Exception_Count : Word;
   //    Connected : Bool;
   //    Connection_ID { ExternalVisible := 'False'} : Word;
   //    MB_State : Word;
   //    TEMP_DATA { ExternalVisible := 'False'} : Array[0..262] of Byte;
   //    Data_Area_Array { S7_SetPoint := 'True'} : Array[1..8] of MB_DataArea;
   //    NDR_immediate : Bool;
   //    DR_immediate : Bool;
   //    BytesReceived : UDInt;
   //    overflow_buffer : Array[0..262] of Byte;
   //    overflow_size_bytes : UInt;
   // END_VAR
BEGIN
END_DATA_BLOCK
